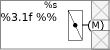
VISUALIZATION SperrAntrieb_MR_Flap_LA_CheckEnabled  // 110x50
VAR_INPUT
    ITF_SPERRANTRIEB_IN   :   ITF_SPERRANTRIEB;
    stExklParameter		:   STRING[40];	
END_VAR
    Frame (61,0 50x50), invisible if: NOT ITF_SPERRANTRIEB_IN.proIsEnabled
        shows Icon_MR_Klappe(ITF_SPERRANTRIEB_IN := ITF_SPERRANTRIEB_IN)
    Frame (0,0 60x25), invisible if: NOT ITF_SPERRANTRIEB_IN.proIsEnabled
        shows ValueUpDwn(ITF_SPERRANTRIEB_IN := ITF_SPERRANTRIEB_IN, uiTextAusrichtung := 6)
    Rectangle (0,0 110x50)
        OnMouseClick:  Dialog=SperrAntrieb_POPUP, Parameters={stExklParameter: stExklParameter, ITF_SPERRANTRIEBIN: ITF_SPERRANTRIEB_IN, uiPopUpGruppe: 0}, OpenCentered=True
END_VISUALIZATION

// 40 Visualizations/ICON/SperrAntrieb_LEFT/Motor_Right/Below/SperrAntrieb_MR_Flap_Txt_L_Below
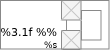
VISUALIZATION SperrAntrieb_MR_Flap_Txt_L_Below  // 110x50
VAR_INPUT
    ITF_SPERRANTRIEB_IN		:   ITF_SPERRANTRIEB;	
END_VAR
VAR_INPUT CONSTANT
    stExklParameter		:   STRING[40] := ' ';	
END_VAR
VAR CONSTANT
	uiIconNr				:	UINT := 3;
END_VAR
    Frame (0,0 110x50), invisible if: NOT fcCheckQuerryReturnIcon(_ITF_In := ITF_SPERRANTRIEB_IN,_uiIconNr_In := uiIconNr)
        shows SperrAntrieb_ML_Flap_LB_CheckQuerry(ITF_SPERRANTRIEB_IN := ITF_SPERRANTRIEB_IN, stExklParameter := stExklParameter)
        shows Icon()
END_VISUALIZATION

// 40 Visualizations/ICON/SperrAntrieb_LEFT/Motor_Right/Below/SperrAntrieb_MR_Flap_LB_CheckQuerry
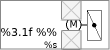
VISUALIZATION SperrAntrieb_MR_Flap_LB_CheckQuerry  // 110x50
VAR_INPUT
    ITF_SPERRANTRIEB_IN   :   ITF_SPERRANTRIEB;
    stExklParameter		:   STRING[40];	
END_VAR
    Frame (0,0 110x50)
        shows SperrAntrieb_ML_Flap_LB_CheckEnabled(ITF_SPERRANTRIEB_IN := ITF_SPERRANTRIEB_IN, stExklParameter := stExklParameter)
END_VISUALIZATION

// 40 Visualizations/ICON/SperrAntrieb_LEFT/Motor_Right/Below/SperrAntrieb_MR_Flap_LB_CheckEnabled
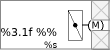
VISUALIZATION SperrAntrieb_MR_Flap_LB_CheckEnabled  // 110x50
VAR_INPUT
    ITF_SPERRANTRIEB_IN   :   ITF_SPERRANTRIEB;
    stExklParameter		:   STRING[40];	
END_VAR
    Frame (61,0 50x50), invisible if: NOT ITF_SPERRANTRIEB_IN.proIsEnabled
        shows Icon_MR_Klappe(ITF_SPERRANTRIEB_IN := ITF_SPERRANTRIEB_IN)
    Frame (0,25 60x25), invisible if: NOT ITF_SPERRANTRIEB_IN.proIsEnabled
        shows ValueDwnUp(ITF_SPERRANTRIEB_IN := ITF_SPERRANTRIEB_IN, uiTextAusrichtung := 6)
    Rectangle (0,0 110x50)
        OnMouseClick:  Dialog=SperrAntrieb_POPUP, Parameters={stExklParameter: , ITF_SPERRANTRIEBIN: ITF_SPERRANTRIEB_IN, uiPopUpGruppe: 0}, OpenCentered=True
END_VISUALIZATION

// 40 Visualizations/ICON/SperrAntrieb_RIGHT/Motor_Left/Above/SperrAntrieb_ML_Flap_Txt_R_Above
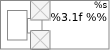
VISUALIZATION SperrAntrieb_ML_Flap_Txt_R_Above  // 110x50
VAR_INPUT
    ITF_SPERRANTRIEB_IN		:   ITF_SPERRANTRIEB;	
END_VAR
VAR_INPUT CONSTANT
    stExklParameter		:   STRING[40] := ' ';	
END_VAR
VAR CONSTANT
	uiIconNr				:	UINT := 6;
END_VAR
    Frame (0,0 110x50), invisible if: NOT fcCheckQuerryReturnIcon(_ITF_In := ITF_SPERRANTRIEB_IN,_uiIconNr_In := uiIconNr)
        shows SperrAntrieb_MR_Flap_RA_CheckQuerry(ITF_SPERRANTRIEB_IN := ITF_SPERRANTRIEB_IN, stExklParameter := stExklParameter)
        shows Icon()
END_VISUALIZATION

// 40 Visualizations/ICON/SperrAntrieb_RIGHT/Motor_Left/Above/SperrAntrieb_ML_Flap_RA_CheckQuerry
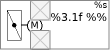
VISUALIZATION SperrAntrieb_ML_Flap_RA_CheckQuerry  // 110x50
VAR_INPUT
    ITF_SPERRANTRIEB_IN   :   ITF_SPERRANTRIEB;
    stExklParameter		:   STRING[40];	
END_VAR
    Frame (0,0 110x50)
        shows SperrAntrieb_MR_Flap_RA_CheckEnabled(ITF_SPERRANTRIEB_IN := ITF_SPERRANTRIEB_IN, stExklParameter := stExklParameter)
END_VISUALIZATION

// 40 Visualizations/ICON/SperrAntrieb_RIGHT/Motor_Left/Above/SperrAntrieb_ML_Flap_RA_CheckEnabled
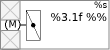
VISUALIZATION SperrAntrieb_ML_Flap_RA_CheckEnabled  // 110x50
VAR_INPUT
    ITF_SPERRANTRIEB_IN   :   ITF_SPERRANTRIEB;
    stExklParameter		:   STRING[40];	
END_VAR
    Frame (0,0 50x50), invisible if: NOT ITF_SPERRANTRIEB_IN.proIsEnabled
        shows Icon_ML_Klappe(ITF_SPERRANTRIEB_IN := ITF_SPERRANTRIEB_IN)
    Frame (50,0 60x25), invisible if: NOT ITF_SPERRANTRIEB_IN.proIsEnabled
        shows ValueUpDwn(ITF_SPERRANTRIEB_IN := ITF_SPERRANTRIEB_IN, uiTextAusrichtung := 4)
    Rectangle (0,0 110x50)
        OnMouseClick:  Dialog=SperrAntrieb_POPUP, Parameters={stExklParameter: stExklParameter, ITF_SPERRANTRIEBIN: ITF_SPERRANTRIEB_IN, uiPopUpGruppe: 0}, OpenCentered=True
END_VISUALIZATION

// 40 Visualizations/ICON/SperrAntrieb_RIGHT/Motor_Left/Below/SperrAntrieb_ML_Flap_Txt_R_Below
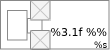
VISUALIZATION SperrAntrieb_ML_Flap_Txt_R_Below  // 110x50
VAR_INPUT
    ITF_SPERRANTRIEB_IN   	:   ITF_SPERRANTRIEB;	
END_VAR
VAR_INPUT CONSTANT
    stExklParameter		:   STRING[40] := ' ';	
END_VAR
VAR CONSTANT
	uiIconNr				:	UINT := 7;
END_VAR
    Frame (0,0 110x50), invisible if: NOT fcCheckQuerryReturnIcon(_ITF_In := ITF_SPERRANTRIEB_IN,_uiIconNr_In := uiIconNr)
        shows SperrAntrieb_MR_Flap_RB_CheckQuerry(ITF_SPERRANTRIEB_IN := ITF_SPERRANTRIEB_IN, stExklParameter := stExklParameter)
        shows Icon()
END_VISUALIZATION

// 40 Visualizations/ICON/SperrAntrieb_RIGHT/Motor_Left/Below/SperrAntrieb_ML_Flap_RB_CheckQuerry
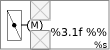
VISUALIZATION SperrAntrieb_ML_Flap_RB_CheckQuerry  // 110x50
VAR_INPUT
    ITF_SPERRANTRIEB_IN   :   ITF_SPERRANTRIEB;
    stExklParameter		:   STRING[40];	
END_VAR
    Frame (0,0 110x50)
        shows SperrAntrieb_MR_Flap_RB_CheckEnabled(ITF_SPERRANTRIEB_IN := ITF_SPERRANTRIEB_IN, stExklParameter := stExklParameter)
END_VISUALIZATION

// 40 Visualizations/ICON/SperrAntrieb_RIGHT/Motor_Left/Below/SperrAntrieb_ML_Flap_RB_CheckEnabled
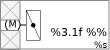
VISUALIZATION SperrAntrieb_ML_Flap_RB_CheckEnabled  // 110x50
VAR_INPUT
    ITF_SPERRANTRIEB_IN   :   ITF_SPERRANTRIEB;
    stExklParameter		:   STRING[40];	
END_VAR
    Frame (0,0 50x50), invisible if: NOT ITF_SPERRANTRIEB_IN.proIsEnabled
        shows Icon_ML_Klappe(ITF_SPERRANTRIEB_IN := ITF_SPERRANTRIEB_IN)
    Frame (50,25 60x25), invisible if: NOT ITF_SPERRANTRIEB_IN.proIsEnabled
        shows ValueDwnUp(ITF_SPERRANTRIEB_IN := ITF_SPERRANTRIEB_IN, uiTextAusrichtung := 4)
    Rectangle (0,0 110x50)
        OnMouseClick:  Dialog=SperrAntrieb_POPUP, Parameters={stExklParameter: , ITF_SPERRANTRIEBIN: ITF_SPERRANTRIEB_IN, uiPopUpGruppe: 0}, OpenCentered=True
END_VISUALIZATION

(* text list Error (id | default | de | en | fr | it)
  0 | keine Meldung Anstehend | Keine Meldung Anstehend | No message pending | Aucun message en attente | Nessun messaggio in sospeso
  1 | Die Abweichung des Stellwertes zum Istwert ist zu hoch | Die Abweichung des Stellwertes zum Istwert ist zu hoch | The deviation of the control value from the actual value is too high /  | L'écart entre la valeur de contrôle et la valeur réelle est trop élevé | Lo scostamento del valore di controllo dal valore effettivo è troppo elevato
  3 | Keine Rückmeldung des Sperrventils beim öffnen | Keine Rückmeldung des Sperrventils beim öffnen | No feedback from the control valve when opening | Pas de retour de la vanne de régulation lors de l'ouverture | Nessun feedback dalla valvola di controllo durante l'apertura
  2 | Keine Rückmeldung des Sperrventils beim schlissen | Keine Rückmeldung des Sperrventils beim schlissen | No feedback from the control valve when closing | Pas de retour de la vanne de régulation lors de la fermeture | Nessun feedback dalla valvola di controllo durante la chiusura
  4 | Leitungsschutzschalter ausfall | Leitungsschutzschalter ausfall | Circuit breaker failure | Défaillance du disjoncteur | Guasto dell'interruttore
  5 | Motorschutzschalter ausfall | Motorschutzschalter ausfall | Motor protection switch failure | Défaillance de l'interrupteur de protection du moteur | Guasto al salvamotore
  6 | Konfigurationsfehler speichern fehlgeschlagen reboot | Konfigurationsfehler speichern fehlgeschlagen reboot | Failed to save configuration error reboot | Impossible d'enregistrer l'erreur de configuration reboot | Impossibile salvare l'errore di configurazione reboot
   |  |  |  |  |  *)

(* text list Info (id | default | de | en | fr | it)
  0 | keine Meldung Anstehend | keine Meldung Anstehend | no message pending | aucun message en attente | nessun messaggio in sospeso
   |  |  |  |  |  *)

(* text list Warnung (id | default | de | en | fr | it)
  0 | Keine Meldung Anstehend | Keine Meldung Anstehend | No message pending | Aucun message en attente | Nessun messaggio in sospeso
  3 | Wahlschalter Hand, Ein | Wahlschalter Hand, Ein | Selector switch hand on | Commutateur de sélection a main, Allumé | Selettore a mano, acceso
  2 | Wahlschalter Hand, Aus | Wahlschalter Hand, Aus | Selector switch hand off | Commutateur de sélection a main, Éteint | Selettore a mano, spento
  1 | Revisionsschalter Ausgeschalten | Revisionsschalter Ausgeschalten | Revision switch off | Commutateur révision Désactiver | Interruttore di revisione disattivato
  4 | Handmodul aktiv | Handmodul aktiv | Hand module active | Module manuel actif | Modulo manuale attivo
   |  |  |  |  |  *)

(* text list KlappenStatus (id | default | Deutsch)
  0 | Gesperrt | Gesperrt
  1 | Schliesst | Schliesst
  2 | ZU | ZU
  3 | Öffnet | Öffnet
  4 | OFFEN | OFFEN
  5 | IDLE | IDLE
   |  |  *)
